FUNCTION_BLOCK FB_Motor
VAR_INPUT
END_VAR
VAR_OUTPUT
END_VAR
VAR
	Up,
	Down,
	Slow ,
	Brake AT %Q* :BOOL;
END_VAR

ACTION MoveDown:
Up:=FALSE;
Down:=TRUE;
Slow:=FALSE;

Brake:=FALSE;
END_ACTION

ACTION MoveUp:
Up:=TRUE;
Down:=FALSE;
Slow:=FALSE;

Brake:=FALSE;
END_ACTION

ACTION SlowDown:
Slow:=TRUE;
END_ACTION

ACTION Stop:
Up:=FALSE;
Down:=FALSE;
Slow:=FALSE;
Brake:=TRUE;
END_ACTION

END_FUNCTION_BLOCK

(* stored: Version 1.1.0.1, ProductVersion 3.1.4024.11
   POU FB_Motor: Id {53cf7bd1-0b81-4de8-baab-b006ee30ff79}, SpecialFunc None
   Action MoveDown: Id {6675dcec-373a-4497-9230-c6e26912dd7e}
   Action MoveUp: Id {c5a4fe86-e2cf-4cb5-9371-4806312c4655}
   Action SlowDown: Id {eb08bf64-661a-4c24-8ae2-baa450dd8056}
   Action Stop: Id {57f754a4-33a4-4431-a0d0-050a24f2b33b} *)
